// Mitsubishi GX Works2 project: 비상버튼 추가 2   PLC: Q02/Q02H

PROGRAM MAIN
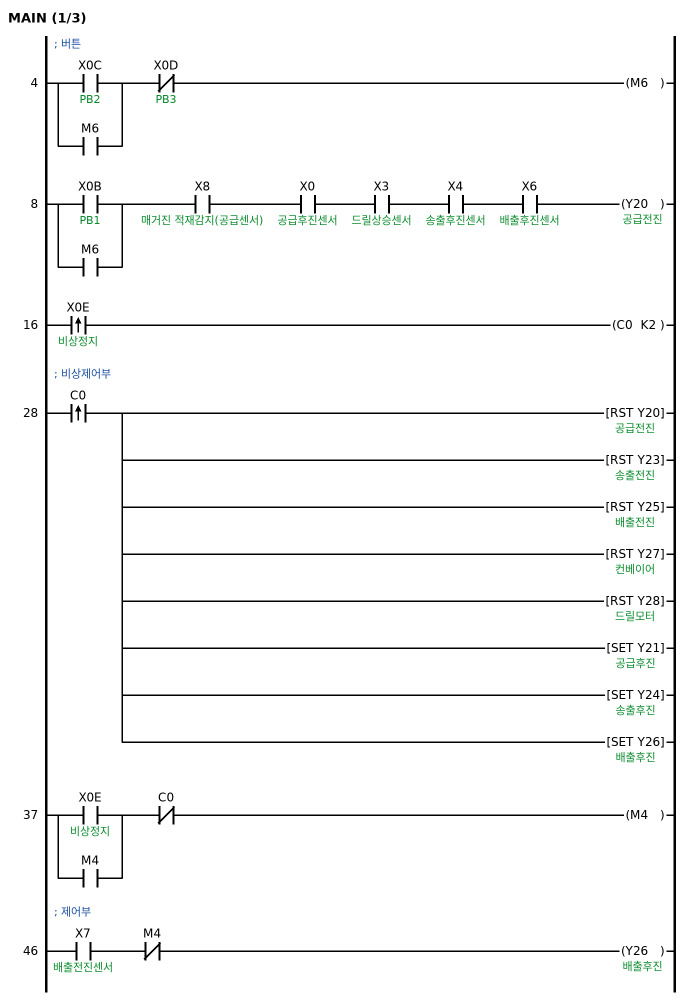
; 버튼
4     LD      X0C  ; PB2
      OR      M6
      ANI     X0D  ; PB3
      OUT     M6
8     LD      X0B  ; PB1
      OR      M6
      AND     X8  ; 매거진 적재감지(공급센서)
      AND     X0  ; 공급후진센서
      AND     X3  ; 드릴상승센서
      AND     X4  ; 송출후진센서
      AND     X6  ; 배출후진센서
      OUT     Y20  ; 공급전진
16    LDP     X0E  ; 비상정지
      OUT     C0 K2
; 비상제어부
28    LDP     C0
      RST     Y20  ; 공급전진
      RST     Y23  ; 송출전진
      RST     Y25  ; 배출전진
      RST     Y27  ; 컨베이어
      RST     Y28  ; 드릴모터
      SET     Y21  ; 공급후진
      SET     Y24  ; 송출후진
      SET     Y26  ; 배출후진
37    LD      X0E  ; 비상정지
      OR      M4
      ANI     C0
      OUT     M4
; 제어부
46    LD      X7  ; 배출전진센서
      ANI     M4
      OUT     Y26  ; 배출후진
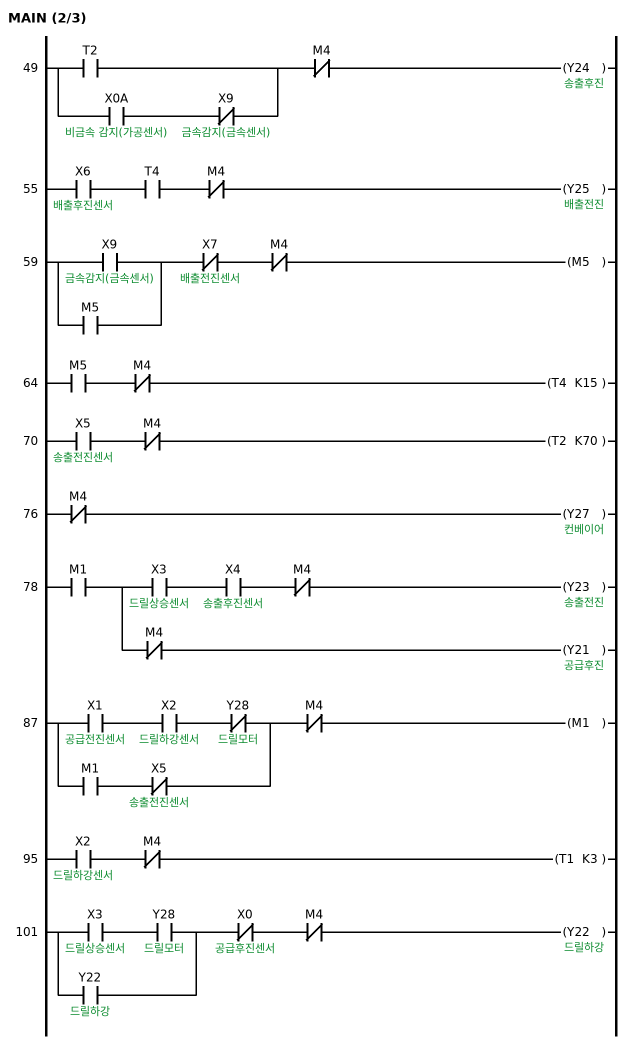
49    LD      T2
      LD      X0A  ; 비금속 감지(가공센서)
      ANI     X9  ; 금속감지(금속센서)
      ORB
      ANI     M4
      OUT     Y24  ; 송출후진
55    LD      X6  ; 배출후진센서
      AND     T4
      ANI     M4
      OUT     Y25  ; 배출전진
59    LD      X9  ; 금속감지(금속센서)
      OR      M5
      ANI     X7  ; 배출전진센서
      ANI     M4
      OUT     M5
64    LD      M5
      ANI     M4
      OUT     T4 K15
70    LD      X5  ; 송출전진센서
      ANI     M4
      OUT     T2 K70
76    LDI     M4
      OUT     Y27  ; 컨베이어
78    LD      M1
      MPS
      AND     X3  ; 드릴상승센서
      AND     X4  ; 송출후진센서
      ANI     M4
      OUT     Y23  ; 송출전진
      MPP
      ANI     M4
      OUT     Y21  ; 공급후진
87    LD      X1  ; 공급전진센서
      AND     X2  ; 드릴하강센서
      ANI     Y28  ; 드릴모터
      LD      M1
      ANI     X5  ; 송출전진센서
      ORB
      ANI     M4
      OUT     M1
95    LD      X2  ; 드릴하강센서
      ANI     M4
      OUT     T1 K3
101   LD      X3  ; 드릴상승센서
      AND     Y28  ; 드릴모터
      OR      Y22  ; 드릴하강
      ANI     X0  ; 공급후진센서
      ANI     M4
      OUT     Y22  ; 드릴하강
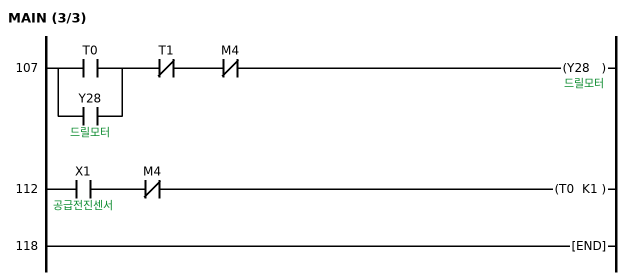
107   LD      T0
      OR      Y28  ; 드릴모터
      ANI     T1
      ANI     M4
      OUT     Y28  ; 드릴모터
112   LD      X1  ; 공급전진센서
      ANI     M4
      OUT     T0 K1
118   END
END_PROGRAM

// device comments not shown above
Y29  ; 적색램프
Y2A  ; 황색램프
Y2B  ; 녹색램프
